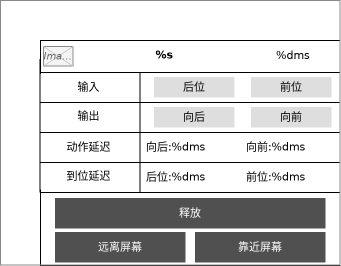
VISUALIZATION Cylinder2  // 341x266
VAR_INPUT
	System:							REFERENCE TO ST_System;
	Cylinder:						REFERENCE TO ST_Cylinder;
	CylinderData:					REFERENCE TO ST_CylinderData;
END_VAR
    RoundedRectangle (40,151 300x115)
    RoundedRectangle (40,40 300x115)
    Rectangle (40,74 300x115)
    Line (40,72) (340,72)
    Rectangle (75,43 179x24), "%s", text variable: Cylinder.arrInfo[System.stMode.eLanguage].sName, input disabled if: Cylinder.stLock.bShield
    Rectangle (258,43 70x25), "%dms", text variable: CylinderData.iAlarmTime, input disabled if: Cylinder.stLock.bShield
        OnMouseClick: write the text variable via VisuDialogs.Numpad
    Line (40,102) (340,102)
    Line (40,132) (340,132)
    Label (41,72 95x30), "输入"
    Label (41,101 95x30), "输出"
    Line (140,192) (140,72)
    RoundedRectangle (154,77 80x20), "后位", colour toggle: Cylinder.stInput.bWork, input disabled if: Cylinder.stLock.bShield
    RoundedRectangle (251,77 80x20), "前位", colour toggle: Cylinder.stInput.bHome, input disabled if: Cylinder.stLock.bShield
    RoundedRectangle (154,107 80x20), "向后", colour toggle: Cylinder.stOutput.bWork, input disabled if: Cylinder.stLock.bShield
    RoundedRectangle (251,107 80x20), "向前", colour toggle: Cylinder.stOutput.bHome, input disabled if: Cylinder.stLock.bShield
    RoundedRectangle (55,198 270x30), "释放", colour toggle: Cylinder.stLock.bOff OR Cylinder.stLock.bAll, input disabled if: Cylinder.stLock.bShield
        tap Cylinder.stControl.stOffRequest.bManual
    RoundedRectangle (55,232 130x30), "远离屏幕", colour toggle: Cylinder.stLock.bWork OR Cylinder.stLock.bAll, input disabled if: Cylinder.stLock.bShield
        tap Cylinder.stControl.stWorkRequest.bManual
    RoundedRectangle (195,232 130x30), "靠近屏幕", colour toggle: Cylinder.stLock.bHome OR Cylinder.stLock.bAll, input disabled if: Cylinder.stLock.bShield
        tap Cylinder.stControl.stHomeRequest.bManual
    Line (340,194) (340,63)
    Line (40,192) (40,59)
    Image (43,46 30x20), image: ImagePool.Cylinder1
    Line (40,162) (340,162)
    Line (40,192) (340,192)
    Label (41,132 95x30), "动作延迟"
    Label (41,161 95x30), "到位延迟"
    RoundedRectangle (143,134 95x26), "向后:%dms", text variable: CylinderData.iWorkRequestTime, input disabled if: Cylinder.stLock.bShield
        OnMouseClick: write the text variable via Default
    RoundedRectangle (243,134 95x26), "向前:%dms", text variable: CylinderData.iHomeRequestTime, input disabled if: Cylinder.stLock.bShield
        OnMouseClick: write the text variable via Default
    RoundedRectangle (143,164 95x26), "后位:%dms", text variable: CylinderData.iWorkDone, input disabled if: Cylinder.stLock.bShield
        OnMouseClick: write the text variable via Default
    RoundedRectangle (243,164 95x26), "前位:%dms", text variable: CylinderData.iHomeDone, input disabled if: Cylinder.stLock.bShield
        OnMouseClick: write the text variable via Default
END_VISUALIZATION

(* stored: Version 1.1.0.1, ProductVersion 3.1.4024.4
   Visu Cylinder2: Id {0240877a-cab1-45ff-ab00-b0e220075aee} *)
